// TIA Portal V18 export
// export: Created 2026-06-08T16:32:21.2470765Z, ExportSetting WithDefaults, DisplayName Totally Integrated Automation Portal, DisplayVersion V18, DisplayName TIA Portal Openness, DisplayVersion V18, DisplayName TIA Portal Version Control Interface, DisplayVersion V18, DisplayName STEP 7 Professional, DisplayVersion V18, DisplayName STEP 7 Safety, DisplayVersion V18, DisplayName WinCC Professional, DisplayVersion V18
FUNCTION_BLOCK "BASE_SORTING_STATION"   // FB8, LAD
VERSION : 0.1
// stored: AutoNumber true, IsIECCheckEnabled false, UDAEnableTagReadback false
BEGIN

REGION Network 1: BEGIN SORTING CONVYER
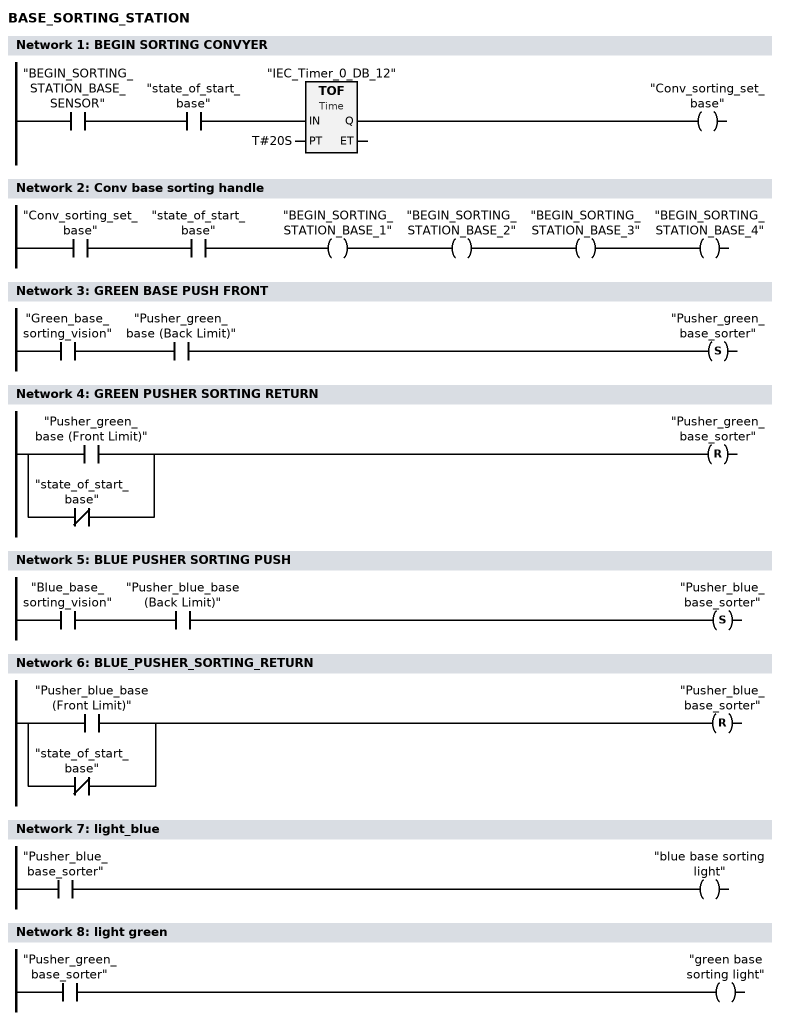
   RUNG wire#powerrail
      Contact( "BEGIN_SORTING_STATION_BASE_SENSOR" )
      Contact( "state_of_start_base" )
      { S7_Templates := "time_type := Time" } "IEC_Timer_0_DB_12".TOF(pt := T#20S, et =>)
      Coil( "Conv_sorting_set_base" )
   END_RUNG
   // the same network as SCL:
   "IEC_Timer_0_DB_12".TOF(IN := "BEGIN_SORTING_STATION_BASE_SENSOR" AND "state_of_start_base", PT := T#20S);
   "Conv_sorting_set_base" := "IEC_Timer_0_DB_12".Q;
END_REGION

REGION Network 2: Conv base sorting handle
   RUNG wire#powerrail
      Contact( "Conv_sorting_set_base" )
      Contact( "state_of_start_base" )
      Coil( "BEGIN_SORTING_STATION_BASE_1" )
      Coil( "BEGIN_SORTING_STATION_BASE_2" )
      Coil( "BEGIN_SORTING_STATION_BASE_3" )
      Coil( "BEGIN_SORTING_STATION_BASE_4" )
   END_RUNG
   // the same network as SCL:
   "BEGIN_SORTING_STATION_BASE_1" := "Conv_sorting_set_base" AND "state_of_start_base";
   "BEGIN_SORTING_STATION_BASE_2" := "BEGIN_SORTING_STATION_BASE_1";
   "BEGIN_SORTING_STATION_BASE_3" := "BEGIN_SORTING_STATION_BASE_1";
   "BEGIN_SORTING_STATION_BASE_4" := "BEGIN_SORTING_STATION_BASE_1";
END_REGION

REGION Network 3: GREEN BASE PUSH FRONT
   RUNG wire#powerrail
      Contact( "Green_base_sorting_vision" )
      Contact( "Pusher_green_base (Back Limit)" )
      S_Coil( "Pusher_green_base_sorter" )
   END_RUNG
   // the same network as SCL:
   IF "Green_base_sorting_vision" AND "Pusher_green_base (Back Limit)" THEN
       "Pusher_green_base_sorter" := TRUE;
   END_IF;
END_REGION

REGION Network 4: GREEN PUSHER SORTING RETURN
   RUNG wire#powerrail
      Contact( "Pusher_green_base (Front Limit)" )
      wire#w1
      R_Coil( "Pusher_green_base_sorter" )
   END_RUNG
   RUNG wire#powerrail
      I_Contact( "state_of_start_base" )
   END_RUNG wire#w1
   // the same network as SCL:
   IF "Pusher_green_base (Front Limit)" OR NOT "state_of_start_base" THEN
       "Pusher_green_base_sorter" := FALSE;
   END_IF;
END_REGION

REGION Network 5: BLUE PUSHER SORTING PUSH
   RUNG wire#powerrail
      Contact( "Blue_base_sorting_vision" )
      Contact( "Pusher_blue_base (Back Limit)" )
      S_Coil( "Pusher_blue_base_sorter" )
   END_RUNG
   // the same network as SCL:
   IF "Blue_base_sorting_vision" AND "Pusher_blue_base (Back Limit)" THEN
       "Pusher_blue_base_sorter" := TRUE;
   END_IF;
END_REGION

REGION Network 6: BLUE_PUSHER_SORTING_RETURN
   RUNG wire#powerrail
      Contact( "Pusher_blue_base (Front Limit)" )
      wire#w1
      R_Coil( "Pusher_blue_base_sorter" )
   END_RUNG
   RUNG wire#powerrail
      I_Contact( "state_of_start_base" )
   END_RUNG wire#w1
   // the same network as SCL:
   IF "Pusher_blue_base (Front Limit)" OR NOT "state_of_start_base" THEN
       "Pusher_blue_base_sorter" := FALSE;
   END_IF;
END_REGION

REGION Network 7: light_blue
   RUNG wire#powerrail
      Contact( "Pusher_blue_base_sorter" )
      Coil( "blue base sorting light" )
   END_RUNG
   // the same network as SCL:
   "blue base sorting light" := "Pusher_blue_base_sorter";
END_REGION

REGION Network 8: light green
   RUNG wire#powerrail
      Contact( "Pusher_green_base_sorter" )
      Coil( "green base sorting light" )
   END_RUNG
   // the same network as SCL:
   "green base sorting light" := "Pusher_green_base_sorter";
END_REGION
END_FUNCTION_BLOCK
